{attribute 'no_explicit_call' := 'FB_EventPublisher is a CLASS and must be accessed using methods or properties'}
FUNCTION_BLOCK EventPublisherWithoutInheritance IMPLEMENTS I_CyclicCall, I_EventPublisher
VAR
	_event							: INT;
	eventPrev						: INT;
	
	observable						: Observable;
END_VAR


// The body of a class must not be used for code.  
// Cyclic code should be called from a method if needed.

METHOD Attach : BOOL
VAR_INPUT
	observer	: I_Observer;
END_VAR
Attach := observable.Attach(observer);
END_METHOD

PROPERTY PUBLIC ChangeEvent : int
SET
// IMPLEMENTED ONLY FOR TESTING PURPOSES
VAR
END_VAR
_event := changeEvent;
END_SET
END_PROPERTY

METHOD CyclicCall
IF eventPrev <> _event 			THEN
	observable.Notify();
	eventPrev := _event;
END_IF
END_METHOD

METHOD Detach : BOOL
VAR_INPUT
	observer	: I_Observer;
END_VAR
Detach := observable.Detach(observer);
END_METHOD

// IMPLEMENTED ONLY FOR TESTING PURPOSES
PROPERTY Event : int
GET
event := _event;
END_GET
END_PROPERTY

END_FUNCTION_BLOCK

(* stored: Version 1.1.0.1, ProductVersion 3.1.4024.11
   POU EventPublisherWithoutInheritance: Id {4c0b0b24-9663-4c35-9fa9-604c8ef8258b}, SpecialFunc None
   Method Attach: Id {c9ce40e8-bcc6-4500-9619-392ddc240421}
   Property ChangeEvent: Id {1c60e725-0b1f-46d6-9aa1-a3f4713694ce}
   Set Set: Id {9205a428-5036-4b6d-9de1-ba82acd6a5db}
   Method CyclicCall: Id {ee124ba0-9538-4355-8558-3d87eeb56a24}
   Method Detach: Id {518a917b-c9bc-4569-aef7-26bf50032e7a}
   Property Event: Id {b8e24b7f-9137-4d0d-b490-03717be08423}
   Get Get: Id {f9412143-d6cb-4b86-8269-e6d6eefff28e} *)
